SUBAPPLICATION Uebung_015a (* Object Pointer umschalten -- 3-fach *)
  (* Standard: 61499-2; Description: Copyright (c) 2023 Meisterschulen am Ostbahnhof This program and the accompanying materials are made available under the terms of the Eclipse Public License 2.0 which is available at https://www.eclipse.org/legal/epl-2.0/ SPDX-License-Identifier: EPL-2.0 *)
  (* Version 1.0, 2023-10-23, Franz Höpfinger, Meisterschulen am Ostbahnhof *)
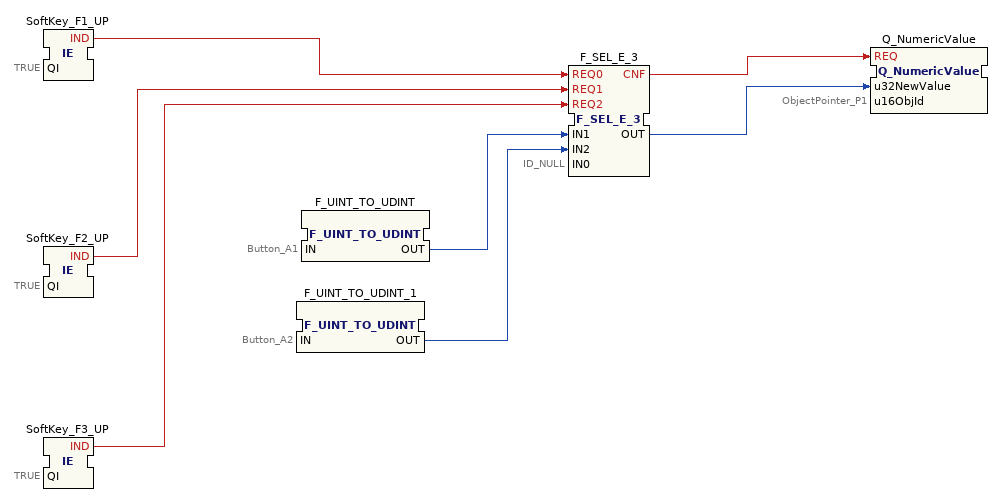
  FBS
    SoftKey_F1_UP : IE(QI := TRUE);
    SoftKey_F2_UP : IE(QI := TRUE);
    F_UINT_TO_UDINT : F_UINT_TO_UDINT(IN := Button_A1);
    F_SEL_E_3 : F_SEL_E_3(IN0 := ID_NULL);
    Q_NumericValue : Q_NumericValue(u16ObjId := ObjectPointer_P1);
    SoftKey_F3_UP : IE(QI := TRUE);
    F_UINT_TO_UDINT_1 : F_UINT_TO_UDINT(IN := Button_A2);
  END_FBS
  EVENT_CONNECTIONS
    F_SEL_E_3.CNF TO Q_NumericValue.REQ;
    SoftKey_F1_UP.IND TO F_SEL_E_3.REQ0;
    SoftKey_F2_UP.IND TO F_SEL_E_3.REQ1;
    SoftKey_F3_UP.IND TO F_SEL_E_3.REQ2;
  END_CONNECTIONS
  DATA_CONNECTIONS
    F_UINT_TO_UDINT.OUT TO F_SEL_E_3.IN1;
    F_SEL_E_3.OUT TO Q_NumericValue.u32NewValue;
    F_UINT_TO_UDINT_1.OUT TO F_SEL_E_3.IN2;
  END_CONNECTIONS
END_SUBAPPLICATION
